(* PLC project Generated.project, CODESYS CODESYS V3.5 SP19 Patch 1 *)
(* stored: creationDateTime 2026-09-14T14:47:22.377047, modificationDateTime 2026-09-14T14:47:22.377047 *)

(* ======================================================================= ST_Modes_Autorisations - Bus public d'autorisations du mode machine ----------------------------------------------------------------------- Doc metier : DOC/AF/AF_Partie-05_Modes_Maintenance_v2.1.md DOC/AF/AF_Partie-02_Architecture_Programme_v3.2.md #2 NC-110 : le prefixe ST_fb* est reserve aux DUT propriete d'un seul FB. Ce DUT est un BUS multi-consommateurs (>=6 domaines : Cycle, Safety, Treuils, Translation, Supervision, Acquisition) -> renomme ST_Modes_Autorisations (bus de domaine public, sans le prefixe FB). Produit par FB_Modes (via PRG_03_Modes_Cycle) Consomme par : Cycle, Safety, Treuils, Translation, Supervision, Acquisition Producteur unique : FB_Modes (via PRG_03_Modes_Cycle) ======================================================================= *)
TYPE ST_Modes_Autorisations : STRUCT
  Mode : E_Mode;  (* Mode arbitre (DISABLE/N1/N2/SEMI_AUTO) *)
  SyncEnable : BOOL;  (* Synchro M1/M2 (logique positive) *)
  InhibitM1 : BOOL;  (* Inhibition M1 (MAINT_N2 only) *)
  InhibitM2 : BOOL;  (* Inhibition M2 (MAINT_N2 only) *)
  JoystickWinchSelectArbitrated : INT;  (* 0=M1+M2 couples nominal, 1=M1, 2=M2 (unitaires MAINT_N2) *)
  CoupledBucketPhaseLocked : BOOL;  (* T248 : phase mouvement couple VERROUILLEE pour ce maintien joystick -> la perte de l'etat ouvert/ferme en mouvement ne relance PAS de correction benne, ni de blocage "descente/montee interdite". Efface au relachement joystick confirme. *)
  WinchSelTransitionHold : BOOL;  (* T248 : changement de selecteur en cours -> requetes mouvement M1/M2 forcees a 0 jusqu'a l'arret confirme (pas de hand-off en mouvement) *)
  HomingApproachEnable : BOOL;  (* Depassement butee haut (N2) *)
  MaintenanceM3TargetEnable : BOOL;  (* Cible Translation Maintenance (N2 only) *)
  ModeChangePendingBlocked : BOOL;  (* AF-05 #4bis - matrice de maintenance Ces trois champs sont des FAITS/DIAGS publies, pas des autorisations : ils restent vrais meme quand le FB est neutralise par Enable=FALSE (etat persistant). Demande de changement de mode REFUSEE : les treuils *)
  ModeChangeBlockReason : STRING(40);  (* ne sont pas a l'arret mecanique confirme (contacteurs retombes ET frein serre ET |v| < seuil). Mode courant maintenu. Motif du blocage de bascule (texte IHM court, ex. "Chgt mode refuse : contacteur M1") *)
  M1ContactorsReleased : BOOL;  (* Détail des 6 sous-conditions de ModeChangeAllowed (diagnostic IHM) — TRUE = condition satisfaite. M1 : contacteurs retombés *)
  M1BrakeApplied : BOOL;  (* M1 : frein serré (NOT M1BrakeIsOpen) *)
  M1SpeedLow : BOOL;  (* M1 : vitesse sous seuil *)
  M2ContactorsReleased : BOOL;  (* M2 : contacteurs retombés *)
  M2BrakeApplied : BOOL;  (* M2 : frein serré (NOT M2BrakeIsOpen) *)
  M2SpeedLow : BOOL;  (* M2 : vitesse sous seuil *)
  HomingRequiredM1 : BOOL;  (* M1 : re-homing obligatoire avant tout retour SEMI_AUTO *)
  HomingRequiredM2 : BOOL;  (* M2 : idem *)
END_STRUCT;
END_TYPE

(* values of E_Mode: DISABLE: Mode Désactivé / Veille de sécurité (sorties bloquées); MAINT_N1: Manuel Niveau 1 : Pilotage unitaire avec toutes sécurités actives; MAINT_N2: Manuel Niveau 2 : Pilotage dégradé (droits étendus + bypasses autorisés); SEMI_AUTO: Mode Semi-Automatique (séquenceur automatique) *)

{attribute 'qualified_only'}
{attribute 'strict'}
TYPE E_Mode : (DISABLE := 0, MAINT_N1 := 1, MAINT_N2 := 2, SEMI_AUTO := 3);
END_TYPE
